TYPE ST_SorterConfig :
{attribute 'OPC.UA.DA' := '1'}
STRUCT
	Name				: STRING[5];
	EquipID				: STRING[5];
	Length				: UINT;
	InductWindow		: UINT;
	MinimumLength		: UINT;
	TailEndLength 		: UINT;
	Output2Offset		: UINT;
	DefaultDestination 	: DINT;
	DefaultDestIdx		: DINT;
	RecircDestination 	: DINT;
	RecircDestIdx 		: DINT;
	RecircUsed			: BOOL;
	RetainOnRestart		: BOOL;
	DivertCount			: DINT;
	RoundRobin			: ST_RoundRobin;
END_STRUCT
END_TYPE

(* stored: Version 1.1.0.1, ProductVersion 3.1.4024.6
   DUT ST_SorterConfig: Id {9ce3f4df-7db1-4bfa-b8ac-5118da50235f} *)
